TYPE st_Rectangulo :
STRUCT
   rASide    	: REAL; // Parámetro de entrada que contiene el lado A del rectangulo.
   rBSide    	: REAL; // Parámetro de entrada que contiene el lado B del rectangulo.	
   rArea		: REAL; // Valor del area
END_STRUCT
END_TYPE

(* stored: Version 1.1.0.1, ProductVersion 3.1.4024.12
   DUT st_Rectangulo: Id {dd70f93a-d982-45c2-b6bc-bd742d42884e} *)
